# B&R Automation Studio project VendingMachine
Automation Studio 4.9

## Configuration ALAB_PPC70

CPU 4PPC70.0702-20B, AutomationRuntime J4.93, Build 4.1.2, Vc V4.73.2

### Task classes (Cpu.sw)
```
Cyclic#1:
  Program <- Program.prg
  Program1 <- Program1.prg
```

### Hardware
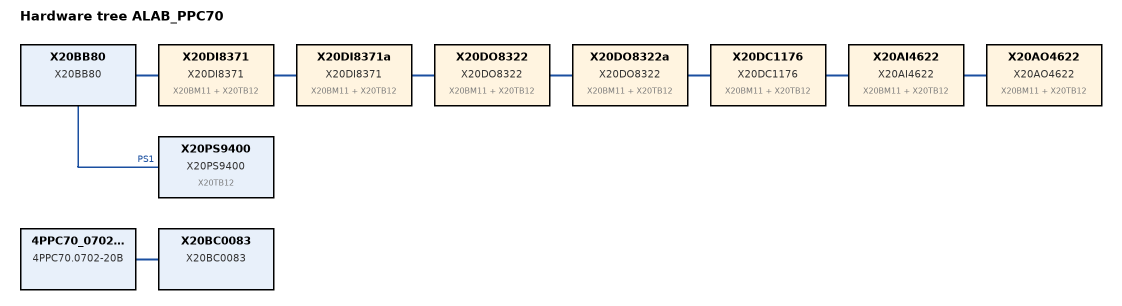
```
4PPC70_0702_20B : 4PPC70.0702-20B v1.5.4.0
  Connector IF2:
    ActivateDevice = 1
    Mode = Manual
    InternetAddress = 192.168.2.20
    SubnetMask = 255.255.255.0
    ActivateSnmp = 2
  ConfigurationID = HTLVB_Sweety_new_ALAB_PPC70
  UserRamSize = 1024
  RemMemSize = 28000
  PermanentPvSize = 2000
  FileDevice1
  FileDeviceName1 = USER
  FileDevicePath1 = USER_PATH
  KeyMappingFile = VC\4PPC70_0702_20B.dis
X20AI4622 : X20AI4622 v1.2.0.0  [SS1 -> X20TB12f.SS; SL -> X20BM11e.SL1]
X20AO4622 : X20AO4622 v1.3.0.0  [SS1 -> X20TB12g.SS; SL -> X20BM11f.SL1]
X20BB80 : X20BB80 v1.1.0.0
X20BC0083 : X20BC0083 v2.14.0.0  [PLK1 -> 4PPC70_0702_20B.IF1 (NodeNumber=1) [Cable Type=PowerlinkCable, Length=10, Version=1.0.0.3]; SL -> X20BB80.SL1]
X20BM11 : X20BM11 v1.1.0.0  [X2X1 -> X20BB80.IF1]
X20BM11a : X20BM11 v1.1.0.0  [X2X1 -> X20BM11.X2X2]
X20BM11b : X20BM11 v1.1.0.0  [X2X1 -> X20BM11a.X2X2]
X20BM11c : X20BM11 v1.1.0.0  [X2X1 -> X20BM11b.X2X2]
X20BM11d : X20BM11 v1.1.0.0  [X2X1 -> X20BM11c.X2X2]
X20BM11e : X20BM11 v1.1.0.0  [X2X1 -> X20BM11d.X2X2]
X20BM11f : X20BM11 v1.1.0.0  [X2X1 -> X20BM11e.X2X2]
X20DC1176 : X20DC1176 v1.4.0.0  [SS1 -> X20TB12e.SS; SL -> X20BM11d.SL1]
X20DI8371 : X20DI8371 v1.4.0.0  [SS1 -> X20TB12a.SS; SL -> X20BM11.SL1]
X20DI8371a : X20DI8371 v1.4.0.0  [SS1 -> X20TB12b.SS; SL -> X20BM11a.SL1]
X20DO8322 : X20DO8322 v1.5.0.0  [SS1 -> X20TB12c.SS; SL -> X20BM11b.SL1]
X20DO8322a : X20DO8322 v1.5.0.0  [SS1 -> X20TB12d.SS; SL -> X20BM11c.SL1]
X20PS9400 : X20PS9400 v1.8.0.0  [SS1 -> X20TB12.SS; PS -> X20BB80.PS1]
X20TB12 : X20TB12 v1.0.0.0
X20TB12a : X20TB12 v1.0.0.0
X20TB12b : X20TB12 v1.0.0.0
X20TB12c : X20TB12 v1.0.0.0
X20TB12d : X20TB12 v1.0.0.0
X20TB12e : X20TB12 v1.0.0.0
X20TB12f : X20TB12 v1.0.0.0
X20TB12g : X20TB12 v1.0.0.0
```

## Configuration Swiity_Automat

CPU X20CP1382, AutomationRuntime G4.83, Build 4.1.2, Vc V4.73.2

### Task classes (Cpu.sw)
```
Cyclic#1:
  Program <- Program.prg
  Program1 <- Program1.prg
VcDataObjects: Visu <- Visu.dob
Binaries: udbdef, vcrt, vcfntttf, FWRules, vccline, vcctext, vccpopup, arial, vccddbox, vcmgr, vccovl, vccnum, vcpfar00, vcdsint, vcpdvnc, vcshared, vcpdsw, vcfile, vcalarm, vcchspot, vccbtn, vccstr, vcgclass, vcdsloc, arialbd, vcnet, Visu02, TCData, vctcal, Visu01, Visu03, vcbclass, vccbmp, iomap, asfw, Role, sysconf, arconfig, ashwd, User, ashwac
Libraries: standard, fileio, asieccon, dataobj, vcresman, astime, AsTCP, dvframe, runtime
```

### Hardware
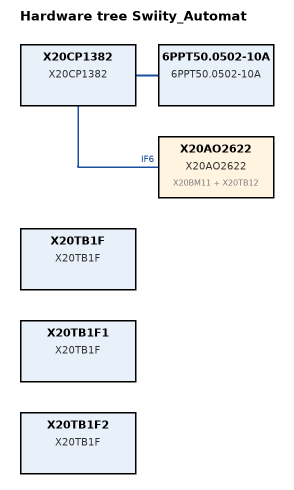
```
6PPT50.0502-10A : 6PPT50.0502-10A v1.3.8.0  [ETH1 -> X20CP1382.IF2 [Cable Type=PowerlinkCable, Length=10, Version=1.0.0.3]]
  Terminal = true
  PasswordVNC = 
  PasswordCIFS = 
  PasswordService = 
  VncVcObjectName = 
  VncAuthentication = 1
  VncPasswordViewOnly = v
  VncPasswordViewControl = c
X20AO2622 : X20AO2622 v1.3.0.0  [SS1 -> X20TB12.SS; SL -> X20BM11.SL1]
X20BM11 : X20BM11 v1.1.0.0  [X2X1 -> X20CP1382.IF6]
X20CP1382 : X20CP1382 v1.14.0.0  [X1 -> X1.SL; X2 -> X2.SL; X3 -> X3.SL]
  Module X1 (Type=X1, Virtual=true, Version=1.14.0.0)
    Connection (Connector=SS1, TargetModule=X20TB1F, TargetConnector=SS)
    Connection (Connector=SL, TargetModule=X20CP1382, TargetConnector=X1)
  Module X2 (Type=X2, Virtual=true, Version=1.14.0.0)
    Connection (Connector=SS1, TargetModule=X20TB1F1, TargetConnector=SS)
    Connection (Connector=SL, TargetModule=X20CP1382, TargetConnector=X2)
  Module X3 (Type=X3, Virtual=true, Version=1.14.0.0)
    Connection (Connector=SS1, TargetModule=X20TB1F2, TargetConnector=SS)
    Connection (Connector=SL, TargetModule=X20CP1382, TargetConnector=X3)
  Connector IF1:
    Baudrate = 115200
    Parity = N
  Connector IF2:
    ActivateDevice = 1
    Mode = Manual
    InternetAddress = 192.168.100.1
    SubnetMask = 255.255.255.0
    Vnc1
    VncVcObjectName1 = Visu
    VncKeyMappingFile1 = VC\PS2-Keyboard1.dis
    VncAuthentication1 = 1
    VncPasswordViewOnly1 = v
    VncPasswordViewControl1 = c
    ActivateSnmp = 2
  Connector IF3:
    Operation = EthOnly
    EthernetMode = DHCPServer
    InternetAddress = 192.168.2.20
    SubnetMask = 255.255.255.0
    ActivateIna = 1
    ActivateANSL = 1
    ActivateSnmp = 2
  ConfigurationID = HTLVB_Zuckerlautomat_Config1
  Simulation = 1
  UserRamSize = 1024
  RemMemSize = 22000
  PermanentPvSize = 8000
X20TB12 : X20TB12 v1.0.0.0
X20TB1F : X20TB1F v1.0.0.0
X20TB1F1 : X20TB1F v1.0.0.0
X20TB1F2 : X20TB1F v1.0.0.0
```

### Cpu.per - X20CP1382/Cpu.per
```iecst
VAR_CONFIG
	Perm_ptMotorX AT %MW0; (* *)
	Perm_preisCent AT %MW8; (* *)
	Perm_muenzwert AT %MW16; (* *)
END_VAR
```

### IoMap.iom - X20CP1382/IoMap.iom
```iecst
VAR_CONFIG
	::aoMotorspeed AT %QW."X20AO2622".AnalogOutput01;
	::diMuenzeinwurf AT %IX."X1".DigitalInput01;
	::doMotor[0] AT %QX."X3".DigitalOutput01;
	::doMotor[1] AT %QX."X3".DigitalOutput02;
	::doMotor[2] AT %QX."X3".DigitalOutput03;
	::doMotor[3] AT %QX."X3".DigitalOutput04;
	doLedEin AT %QX."X3".DigitalOutput05;
END_VAR
```

## Logical view

Binary libraries used (declarations not repeated): operator, runtime, astime, AsIecCon, standard

### Global.typ - Global data types
```iecst
TYPE
	eVisuPages :
		(
		_00_Init := 0,
		_10_Main := 10,
		_15_Zahlungsart := 15,
		_20_BarBezahlen := 20,
		_30_KarteBezahlen := 30,
		_40_Ausgabe := 40,
		_50_Danke := 50,
		_90_Fehler := 90,
		_900_Settings0 := 900,
		_910_Settings1 := 910
		);
	tVisu_buttons : 	STRUCT
		P10_Selection1 : USINT;
		P10_Selection2 : USINT;
		P10_Selection3 : USINT;
		P10_Selection4 : USINT;
		P10_StartQuiz : USINT;
		P910_MoveMotor : USINT;
		PXX_GotoSettings : USINT;
		PXX_SettingsNextPage : USINT;
		PXX_SettingsPrevPage : USINT;
		P10_WaehleBar : USINT;
		P10_WaehleKarte : USINT;
		P20_BestaetigeBar : USINT;
		P30_BestaetigeKarte : USINT;
		PXX_Abbrechen : USINT;
	END_STRUCT;
	tVisu_settings : 	STRUCT
		Language : USINT;
		Language_Updated : BOOL;
		actMotorSelected : INT;
		actMotorSelected_Updated : BOOL;
		ptMotorVisuInput : INT;
		ptMotorX : ARRAY[0..3]OF INT;
		ptMotorX_Updated : BOOL;
		Text_Selection_de : ARRAY[0..3]OF STRING[80];
		Text_Selection_en : ARRAY[0..3]OF STRING[80];
		Text_Selection_Visu : ARRAY[0..3]OF STRING[80];
		Text_Selection_Visu_Updated : ARRAY[0..3]OF BOOL;
	END_STRUCT;
	tVisu : 	STRUCT
		page : tVisu_page;
		buttons : tVisu_buttons;
		settings : tVisu_settings;
	END_STRUCT;
	tVisu_page : 	STRUCT
		setpage : eVisuPages;
		actpage : eVisuPages;
	END_STRUCT;
	tFach : 	STRUCT
		abstandCm : UINT;
		istLeer : BOOL;
		referenzCm : UINT;
		preisCent : UINT;
		name : STRING[20];
	END_STRUCT;
	tAuswahl : 	STRUCT
		fachNr : UINT;
		aktiv : BOOL;
		preisCent : UINT;
	END_STRUCT;
	tZahlung : 	STRUCT
		modus : UINT;
		eingezahltCent : UINT;
		status : UINT;
		startZeitMs : UDINT;
		bezahltGenug : BOOL;
	END_STRUCT;
	tNfcInfo : 	STRUCT
		uidHex : STRING[20];
		zeitstempelMs : UDINT;
		erkannt : USINT;
		inWhitelist : USINT;
		wartet : USINT;
	END_STRUCT;
	tMuenze : 	STRUCT
		impulse : UDINT;
		summeCent : UINT;
		wertProImpulsCent : UINT;
		letzterImpulsMs : UDINT;
	END_STRUCT;
END_TYPE
```

### Global.var - Global variables
```iecst
VAR
	Visu : tVisu;
	aoMotorspeed : INT;
	diMuenzeinwurf : BOOL;
	doMotor : ARRAY[0..3] OF BOOL;
	doLedEin : BOOL;
	psMotorspeed : INT;
	gFach : ARRAY[0..3] OF tFach;
	gSel : tAuswahl;
	gPay : tZahlung;
	gNfc : tNfcInfo;
	gCoin : tMuenze;
	do_Relais : BOOL;
	diEspFach : ARRAY[0..3] OF BOOL;
	diEspNfc : BOOL;
	Perm_motorLaufzeit : ARRAY[0..3] OF UINT;
END_VAR
VAR RETAIN
	Perm_ptMotorX : ARRAY[0..3] OF INT;
	Perm_preisCent : ARRAY[0..3] OF UINT;
	Perm_muenzwert : UINT;
END_VAR
VAR CONSTANT
	TIMEOUT_ZAHLUNG_MS : UDINT := 60000;
END_VAR
```

### Package Logical/Libraries - Global libraries

- Visualisation Logical/Visu (not shown)

### Program Logical/Program (ANSIC) - Snackomat Hauptlogik (TCP zu ESP32)

#### Variables.var
```iecst
VAR
	stateZahlung : UINT;
	lastMotorReqMs : UDINT;
	jetztMs : UDINT;
	iFach : USINT;
	settingsHoldStartMs : UDINT;
	settingsHoldActive : BOOL;
	iTextSel : USINT;
END_VAR
```

#### Cyclic.cpp
```cpp
/* ============================================================
 * Snackomat Hauptprogramm - Cyclic
 *
 * Fach-Status und NFC werden ueber 5 direkte Digitaleingaenge
 * vom ESP32 gelesen:
 *   diEspFach[0..3] : HIGH = VOLL, LOW = LEER
 *   diEspNfc        : HIGH (~2s) = Karte erkannt (beliebige Karte)
 *
 * Motorsteuerung: PLC schaltet doMotor[] direkt nach Ablauf von
 * Perm_motorLaufzeit[].
 * ========================================================== */

#include <bur/plctypes.h>
#include <string.h>
#include <stdlib.h>
#include <stdio.h>

#ifdef _DEFAULT_INCLUDES
	#include <AsDefault.h>
#endif

unsigned long bur_heap_size = 0xFFFF;

/* Fach-Button gedrueckt? Liefert 1..4 oder 0 */
static UINT pruefeFachButton(void)
{
	if (Visu.buttons.P10_Selection1) { Visu.buttons.P10_Selection1 = 0; return 1; }
	if (Visu.buttons.P10_Selection2) { Visu.buttons.P10_Selection2 = 0; return 2; }
	if (Visu.buttons.P10_Selection3) { Visu.buttons.P10_Selection3 = 0; return 3; }
	if (Visu.buttons.P10_Selection4) { Visu.buttons.P10_Selection4 = 0; return 4; }
	return 0;
}

void _CYCLIC ProgramCyclic(void)
{
	UINT fach;
	UINT idx;
	USINT i;

	jetztMs = jetztMs + 10;

	/* ====================================================
	 * Digitaleingaenge vom ESP32 auslesen
	 * ==================================================== */
	for (i = 0; i < 4; i++) {
		gFach[i].istLeer = diEspFach[i] ? 0 : 1;   /* LOW = LEER */
	}
	gNfc.erkannt     = diEspNfc ? 1 : 0;
	gNfc.inWhitelist = diEspNfc ? 1 : 0;   /* jede Karte gueltig */
	gNfc.wartet      = diEspNfc ? 0 : 1;

	/* Hilfsvariable fuer Visu: Farbwechsel der Progress-Bar */
	gPay.bezahltGenug = (gCoin.summeCent >= gSel.preisCent && gSel.aktiv) ? 1 : 0;

	/* ====================================================
	 * Start-Screen: _00_Init 3 Sekunden zeigen,
	 * dann automatisch auf _10_Main wechseln
	 * ==================================================== */
	if (Visu.page.actpage == _00_Init && jetztMs >= 3000) {
		Visu.page.setpage = _10_Main;
	}

	/* ====================================================
	 * Lang-Druck auf PXX_GotoSettings (2s) -> Settings-Seite
	 * ==================================================== */
	if (Visu.buttons.PXX_GotoSettings) {
		if (!settingsHoldActive) {
			settingsHoldActive  = 1;
			settingsHoldStartMs = jetztMs;
		} else if ((jetztMs - settingsHoldStartMs) >= 2000) {
			Visu.buttons.PXX_GotoSettings = 0;
			settingsHoldActive            = 0;
			Visu.page.setpage             = _900_Settings0;
		}
	} else {
		settingsHoldActive = 0;
	}

	/* Aus Settings raus: Prev/Next-Buttons zwischen 900/910, Abbrechen -> Main */
	if (Visu.buttons.PXX_SettingsNextPage || Visu.buttons.PXX_SettingsPrevPage) {
		Visu.buttons.PXX_SettingsNextPage = 0;
		Visu.buttons.PXX_SettingsPrevPage = 0;
		if (Visu.page.actpage == _900_Settings0)       Visu.page.setpage = _910_Settings1;
		else if (Visu.page.actpage == _910_Settings1)  Visu.page.setpage = _900_Settings0;
	}

	/* ====================================================
	 * Settings-Logik (nur aktiv auf Seite 910)
	 * Motor manuell tippbetreiben + Motorzeit pro Fach speichern
	 * ==================================================== */
	if (Visu.page.actpage == _910_Settings1) {
		USINT selIdx = (USINT) Visu.settings.actMotorSelected;
		if (selIdx > 3) selIdx = 0;

		/* Tippbetrieb: gedrueckt -> Motor an */
		if (Visu.buttons.P910_MoveMotor) {
			doMotor[selIdx] = 1;
			aoMotorspeed    = psMotorspeed;
		} else {
			doMotor[selIdx] = 0;
			aoMotorspeed    = 0;
		}

		/* Zeiteingabe aus Visu -> Perm speichern */
		if (Visu.settings.ptMotorX_Updated) {
			Visu.settings.ptMotorX_Updated = 0;
			Visu.settings.ptMotorX[selIdx] = Visu.settings.ptMotorVisuInput;
			Perm_ptMotorX[selIdx]          = Visu.settings.ptMotorVisuInput;
			Perm_motorLaufzeit[selIdx]     = (UINT) Visu.settings.ptMotorVisuInput;
		}

		/* Motor-Auswahl gewechselt -> aktuelle Zeit auf Visu schreiben */
		if (Visu.settings.actMotorSelected_Updated) {
			Visu.settings.actMotorSelected_Updated = 0;
			Visu.settings.ptMotorVisuInput = Visu.settings.ptMotorX[selIdx];
		}
	}

	/* ====================================================
	 * Sprach-Umschaltung (de/en)
	 * ==================================================== */
	if (Visu.settings.Language_Updated) {
		for (iTextSel = 0; iTextSel < 4; iTextSel++) {
			if (Visu.settings.Language == 0) {
				strcpy(Visu.settings.Text_Selection_Visu[iTextSel],
				       Visu.settings.Text_Selection_en[iTextSel]);
			} else {
				strcpy(Visu.settings.Text_Selection_Visu[iTextSel],
				       Visu.settings.Text_Selection_de[iTextSel]);
			}
		}
		Visu.settings.Language_Updated = 0;
	}

	/* Texteingabe aus Visu -> in entsprechenden Sprachspeicher */
	for (iTextSel = 0; iTextSel < 4; iTextSel++) {
		if (Visu.settings.Text_Selection_Visu_Updated[iTextSel]) {
			Visu.settings.Text_Selection_Visu_Updated[iTextSel] = 0;
			if (Visu.settings.Language == 0) {
				strcpy(Visu.settings.Text_Selection_en[iTextSel],
				       Visu.settings.Text_Selection_Visu[iTextSel]);
			} else {
				strcpy(Visu.settings.Text_Selection_de[iTextSel],
				       Visu.settings.Text_Selection_Visu[iTextSel]);
			}
			strncpy(gFach[iTextSel].name,
			        Visu.settings.Text_Selection_Visu[iTextSel], 19);
			gFach[iTextSel].name[19] = 0;
		}
	}

	/* ====================================================
	 * Abbrechen-Button
	 * ==================================================== */
	if (Visu.buttons.PXX_Abbrechen) {
		Visu.buttons.PXX_Abbrechen = 0;
		stateZahlung      = 0;
		gPay.modus        = 0;
		gPay.status       = 2;
		gCoin.summeCent   = 0;
		gCoin.impulse     = 0;
		gSel.aktiv        = 0;
		gSel.fachNr       = 0;
		Visu.page.setpage = _10_Main;
	}

	/* ====================================================
	 * Zahlungs-State-Machine
	 * ==================================================== */
	switch (stateZahlung) {

	case 0: /* idle */
		fach = pruefeFachButton();
		if (fach > 0) {
			idx = fach - 1;
			if (gFach[idx].istLeer) {
				gPay.status       = 3;
				Visu.page.setpage = _90_Fehler;
			} else {
				gSel.fachNr       = fach;
				gSel.preisCent    = gFach[idx].preisCent;
				gSel.aktiv        = 1;
				gPay.startZeitMs  = jetztMs;
				stateZahlung      = 1;
				Visu.page.setpage = _15_Zahlungsart;
			}
		}
		break;

	case 1: /* Bar oder Karte? */
		if (Visu.buttons.P10_WaehleBar) {
			Visu.buttons.P10_WaehleBar = 0;
			gPay.modus        = 1;
			stateZahlung      = 2;
			Visu.page.setpage = _20_BarBezahlen;
		} else if (Visu.buttons.P10_WaehleKarte) {
			Visu.buttons.P10_WaehleKarte = 0;
			gPay.modus        = 2;
			stateZahlung      = 3;
			Visu.page.setpage = _30_KarteBezahlen;
		}
		if ((jetztMs - gPay.startZeitMs) > TIMEOUT_ZAHLUNG_MS) {
			stateZahlung      = 0;
			gPay.modus        = 0;
			gPay.status       = 2;
			gCoin.summeCent   = 0;
			gCoin.impulse     = 0;
			gSel.aktiv        = 0;
			gSel.fachNr       = 0;
			Visu.page.setpage = _10_Main;
		}
		break;

	case 2: /* Bar */
		gPay.eingezahltCent = gCoin.summeCent;
		if (gCoin.summeCent >= gSel.preisCent
		    && Visu.buttons.P20_BestaetigeBar) {
			Visu.buttons.P20_BestaetigeBar = 0;
			stateZahlung     = 6;
			lastMotorReqMs   = jetztMs;
		}
		if ((jetztMs - gPay.startZeitMs) > TIMEOUT_ZAHLUNG_MS) {
			stateZahlung      = 0;
			gPay.modus        = 0;
			gPay.status       = 2;
			gCoin.summeCent   = 0;
			gCoin.impulse     = 0;
			gSel.aktiv        = 0;
			gSel.fachNr       = 0;
			Visu.page.setpage = _10_Main;
		}
		break;

	case 3: /* Karte - warten auf NFC-Eingang + Bestaetigung */
		if (gNfc.erkannt && gNfc.inWhitelist
		    && Visu.buttons.P30_BestaetigeKarte) {
			Visu.buttons.P30_BestaetigeKarte = 0;
			stateZahlung   = 6;
			lastMotorReqMs = jetztMs;
		}
		if ((jetztMs - gPay.startZeitMs) > TIMEOUT_ZAHLUNG_MS) {
			stateZahlung      = 0;
			gPay.modus        = 0;
			gPay.status       = 2;
			gCoin.summeCent   = 0;
			gCoin.impulse     = 0;
			gSel.aktiv        = 0;
			gSel.fachNr       = 0;
			Visu.page.setpage = _10_Main;
		}
		break;

	case 6: /* Motor-Start */
		idx = gSel.fachNr - 1;
		if (idx <= 3) doMotor[idx] = 1;
		stateZahlung      = 4;
		lastMotorReqMs    = jetztMs;
		Visu.page.setpage = _40_Ausgabe;
		break;

	case 4: /* Motor laeuft - Timer-basiertes Stoppen */
		idx = gSel.fachNr - 1;
		if (idx <= 3 && (jetztMs - lastMotorReqMs) >= (UDINT) Perm_motorLaufzeit[idx]) {
			doMotor[idx]      = 0;
			gPay.status       = 1;
			stateZahlung      = 5;
			lastMotorReqMs    = jetztMs;
			Visu.page.setpage = _50_Danke;
		}
		/* Safety-Timeout */
		if ((jetztMs - lastMotorReqMs) > 8000) {
			if (idx <= 3) doMotor[idx] = 0;
			gPay.status       = 3;
			stateZahlung      = 0;
			Visu.page.setpage = _90_Fehler;
		}
		break;

	case 5: /* Danke-Screen 5.5s zeigen */
		if ((jetztMs - lastMotorReqMs) > 5500) {
			stateZahlung      = 0;
			gPay.modus        = 0;
			gPay.status       = 0;
			gCoin.summeCent   = 0;
			gCoin.impulse     = 0;
			gSel.aktiv        = 0;
			gSel.fachNr       = 0;
			Visu.page.setpage = _10_Main;
		}
		break;
	}

	Visu.page.actpage = Visu.page.setpage;
	do_Relais = (stateZahlung == 4);

	(void) iFach;
}
```

#### Init.cpp
```cpp
/* ============================================================
 * Snackomat Hauptprogramm - Init
 * ========================================================== */

#include <bur/plctypes.h>
#include <string.h>

#ifdef _DEFAULT_INCLUDES
	#include <AsDefault.h>
#endif

void _INIT ProgramInit(void)
{
	USINT i;

	if (Perm_muenzwert == 0) Perm_muenzwert = 10;
	for (i = 0; i < 4; i++) {
		if (Perm_preisCent[i] == 0)     Perm_preisCent[i]     = 150;
		if (Perm_motorLaufzeit[i] == 0) Perm_motorLaufzeit[i] = 2500;
	}

	for (i = 0; i < 4; i++) {
		gFach[i].abstandCm  = 0;
		gFach[i].istLeer    = 0;
		gFach[i].referenzCm = 0;
		gFach[i].preisCent  = Perm_preisCent[i];
	}
	strcpy(gFach[0].name, "Produkt 1");
	strcpy(gFach[1].name, "Produkt 2");
	strcpy(gFach[2].name, "Produkt 3");
	strcpy(gFach[3].name, "Produkt 4");

	for (i = 0; i < 4; i++) {
		Visu.settings.ptMotorX[i] = (INT) Perm_ptMotorX[i];
	}
	Visu.settings.ptMotorVisuInput = (INT) Perm_ptMotorX[0];

	gSel.fachNr = 0;     gSel.aktiv = 0;     gSel.preisCent = 0;
	gPay.modus  = 0;     gPay.eingezahltCent = 0;    gPay.status = 0;
	gNfc.erkannt = 0;    gNfc.inWhitelist = 0;
	gCoin.impulse = 0;   gCoin.summeCent = 0;   gCoin.wertProImpulsCent = Perm_muenzwert;

	Visu.page.setpage = _00_Init;
	Visu.page.actpage = _00_Init;

	stateZahlung = 0;
}
```

### Program Logical/Program1 (ANSIC) - Muenzzaehlung

#### Cyclic.cpp - Cyclic code
```cpp
/* ============================================================
 * Muenzzaehlung (Program1) - Cyclic
 *
 * Liest diMuenzeinwurf (X20 DI), erkennt steigende Flanken und
 * addiert pro Impuls den Wert aus gCoin.wertProImpulsCent zu
 * gCoin.summeCent.
 * ========================================================== */

#include <bur/plctypes.h>

#ifdef _DEFAULT_INCLUDES
	#include <AsDefault.h>
#endif

unsigned long bur_heap_size = 0xFFFF;

void _CYCLIC ProgramCyclic(void)
{
	/* einfacher Zyklus-Zaehler (10 ms pro Tick) */
	static UDINT counter = 0;
	counter += 10;

	/* Steigende Flanke an Lichtschranke (=diMuenzeinwurf)? */
	if (diMuenzeinwurf && !lastInput) {
		/* Entprellung: nur zaehlen wenn > entprellungMs seit letzter Flanke */
		if ((counter - lastEdgeMs) > entprellungMs) {
			gCoin.impulse++;
			gCoin.summeCent       += gCoin.wertProImpulsCent;
			gCoin.letzterImpulsMs  = counter;
			lastEdgeMs             = counter;
		}
	}
	lastInput = diMuenzeinwurf;
}
```

#### Init.cpp - Initialization code
```cpp
/* ============================================================
 * Muenzzaehlung (Program1) - Init
 * ========================================================== */
#include <bur/plctypes.h>

#ifdef _DEFAULT_INCLUDES
	#include <AsDefault.h>
#endif

void _INIT ProgramInit(void)
{
	lastInput     = 0;
	lastEdgeMs    = 0;
}
```

#### Exit.cpp - Exit code
```cpp
#include <bur/plctypes.h>

#ifdef _DEFAULT_INCLUDES
	#include <AsDefault.h>
#endif

void _EXIT ProgramExit(void)
{
	// Insert code here

}
```

#### Variables.var - Local variables
```iecst
(* ========================================================== *)
(* Muenzzaehlung (Program1) - lokale Variablen                *)
(* Zaehlt Impulse der Lichtschranke (di_Lichtschranke)        *)
(* mit Entprellung.                                           *)
(* ========================================================== *)

VAR

    lastInput       : BOOL;          (* Zustand im letzten Tick *)
    lastEdgeMs      : UDINT;         (* Zeitpunkt letzter steigender Flanke *)
    entprellungMs   : UDINT := 20;   (* 20ms Entprellung *)

END_VAR

VAR CONSTANT

END_VAR
```

Listed in the project but not available here: Logical/Program1/Types.typ
